KUKA KRL program: Weld_PartA.src, Weld_PartA.dat

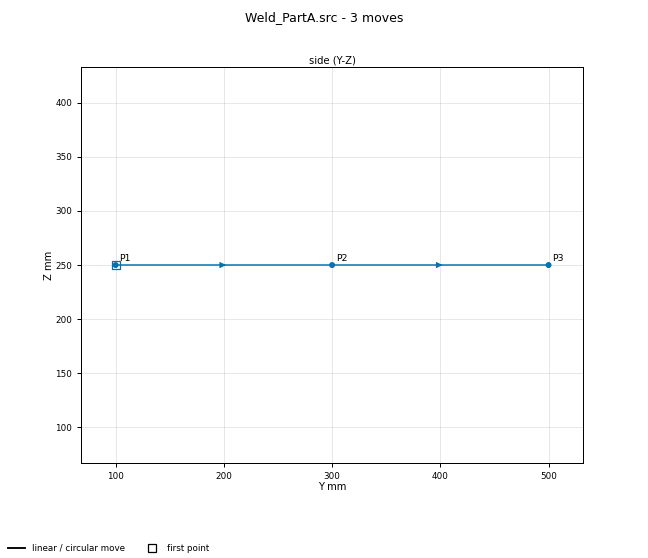
[picture p0: tool path of Weld_PartA.src, 3 of 5 moves have a stored position in this frame; points joined in program order, loops and branches not executed]
--- Weld_PartA.src ---
&ACCESS RVP
&REL 1
&COMMENT Han suon xe Wave Alpha
DEF Weld_PartA()
  ;FOLD INI
    ;FOLD BASISTECH INI
      BAS(#INITMOV, 0)
    ;ENDFOLD
  ;ENDFOLD

  PTP HOME Vel=100% DEFAULT

  LIN P1
  LIN P2
  LIN P3

  PTP HOME Vel=100% DEFAULT

END

--- Weld_PartA.dat ---
&ACCESS RV
&REL 1
DEFDAT Weld_PartA PUBLIC
  DECL E6POS HOME={A1 0.0, A2 -90.0, A3 90.0, A4 0.0, A5 0.0, A6 0.0}
  DECL E6POS P1={X 400.0, Y 100.0, Z 250.0, A 0.0, B 90.0, C 0.0, S 2, T 10}
  DECL E6POS P2={X 400.0, Y 300.0, Z 250.0, A 0.0, B 90.0, C 0.0, S 2, T 10}
  DECL E6POS P3={X 400.0, Y 500.0, Z 250.0, A 0.0, B 90.0, C 0.0, S 2, T 10}
ENDDAT
